// Mitsubishi GX Works2 project: 곱하기   PLC: Q02/Q02H

PROGRAM MAIN
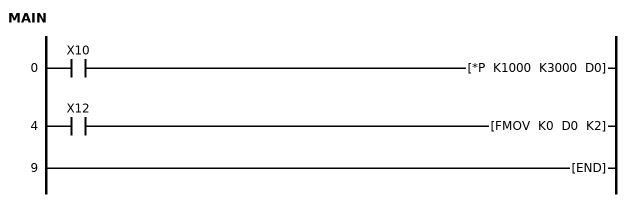
0     LD      X10
      *P      K1000 K3000 D0
4     LD      X12
      FMOV    K0 D0 K2
9     END
END_PROGRAM
